FUNCTION_BLOCK bfb_monday_classifier
  (* Standard: 61499-2 *)
  (* Version 0.1, 2018-00-07, hpea485, UOA *)
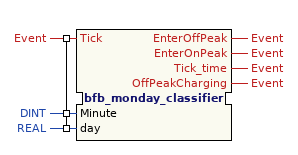
  EVENT_INPUT
    Tick WITH Minute, day;
  END_EVENT
  EVENT_OUTPUT
    EnterOffPeak;
    EnterOnPeak;
    Tick_time;
    OffPeakCharging;
  END_EVENT
  VAR_INPUT
    Minute : DINT;
    day : REAL;
  END_VAR
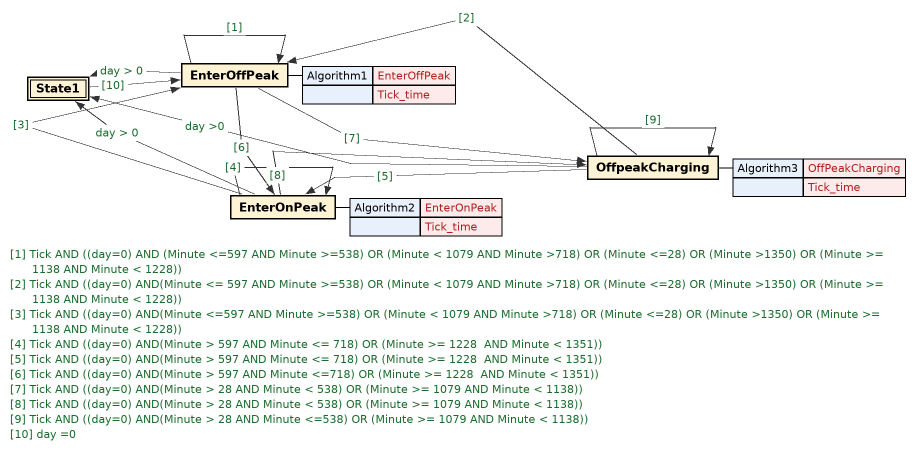
  EC_STATES
    State1;
    EnterOffPeak : Algorithm1 -> EnterOffPeak, -> Tick_time;
    EnterOnPeak : Algorithm2 -> EnterOnPeak, -> Tick_time;
    OffpeakCharging : Algorithm3 -> OffPeakCharging, -> Tick_time;
  END_STATES
  EC_TRANSITIONS
    EnterOffPeak TO EnterOffPeak := Tick AND ((day=0) AND (Minute <=597 AND Minute >=538) OR (Minute < 1079 AND Minute >718) OR (Minute <=28) OR (Minute >1350) OR (Minute >= 1138 AND Minute < 1228));
    EnterOffPeak TO EnterOnPeak := Tick AND ((day=0) AND(Minute > 597 AND Minute <=718) OR (Minute >= 1228  AND Minute < 1351));
    EnterOffPeak TO OffpeakCharging := Tick AND ((day=0) AND(Minute > 28 AND Minute < 538) OR (Minute >= 1079 AND Minute < 1138));
    EnterOffPeak TO State1 := day > 0;
    EnterOnPeak TO EnterOffPeak := Tick AND ((day=0) AND(Minute <=597 AND Minute >=538) OR (Minute < 1079 AND Minute >718) OR (Minute <=28) OR (Minute >1350) OR (Minute >= 1138 AND Minute < 1228));
    EnterOnPeak TO EnterOnPeak := Tick AND ((day=0) AND(Minute > 597 AND Minute <= 718) OR (Minute >= 1228  AND Minute < 1351));
    EnterOnPeak TO OffpeakCharging := Tick AND ((day=0) AND(Minute > 28 AND Minute < 538) OR (Minute >= 1079 AND Minute < 1138));
    EnterOnPeak TO State1 := day > 0;
    OffpeakCharging TO OffpeakCharging := Tick AND ((day=0) AND(Minute > 28 AND Minute <=538) OR (Minute >= 1079 AND Minute < 1138));
    OffpeakCharging TO EnterOnPeak := Tick AND ((day=0) AND(Minute > 597 AND Minute <= 718) OR (Minute >= 1228  AND Minute < 1351));
    OffpeakCharging TO EnterOffPeak := Tick AND ((day=0) AND(Minute <= 597 AND Minute >=538) OR (Minute < 1079 AND Minute >718) OR (Minute <=28) OR (Minute >1350) OR (Minute >= 1138 AND Minute < 1228));
    OffpeakCharging TO State1 := day >0;
    State1 TO EnterOffPeak := day =0;
  END_TRANSITIONS
  ALGORITHM Algorithm1 IN C:
printf("Entered OFF PEAK.....\r\n");
  END_ALGORITHM
  ALGORITHM Algorithm2 IN C:
printf(" Entered On peak .....\r\n ");
  END_ALGORITHM
  ALGORITHM Algorithm3 IN C:
printf(" OffPeak Charging \r\n ");
  END_ALGORITHM
END_FUNCTION_BLOCK
